// SIMATIC S7-200 project (STEP 7-Micro/WIN), CPU 224 CN REL 02.01

ORGANIZATION_BLOCK 主程序:OB1
TITLE=程序注释
BEGIN
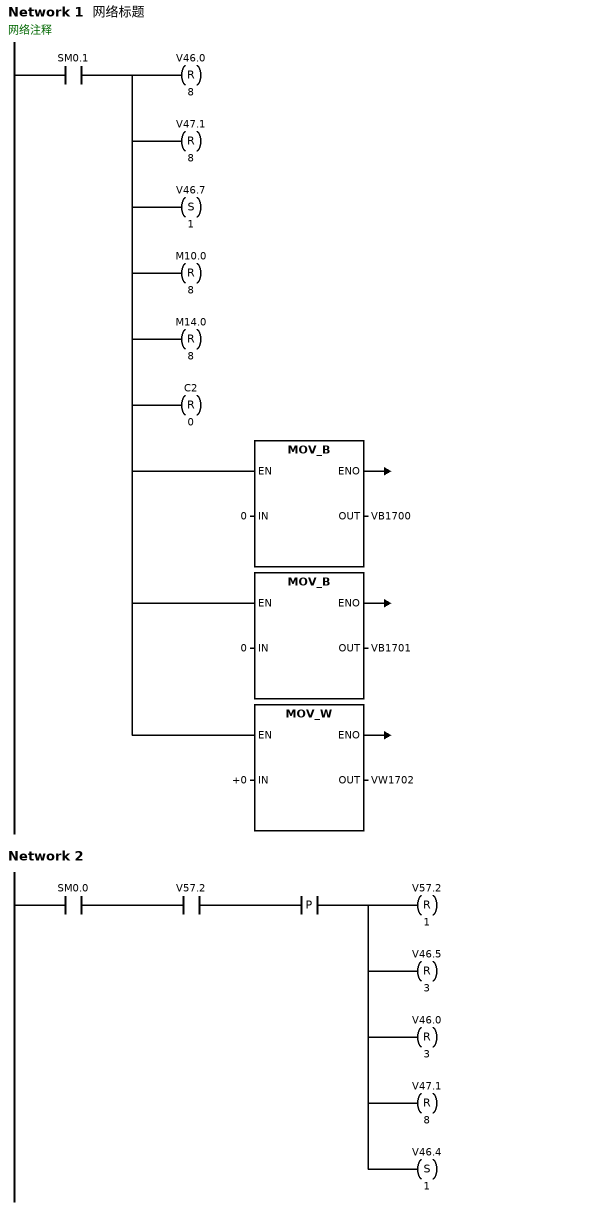
Network 1 // 网络标题
// 网络注释
LD     SM0.1
R      V46.0, 8
R      V47.1, 8
S      V46.7, 1
R      M10.0, 8
R      M14.0, 8
R      C2, 0
MOVB   0, VB1700
MOVB   0, VB1701
MOVW   +0, VW1702
Network 2
LD     SM0.0
A      V57.2
EU
R      V57.2, 1
R      V46.5, 3
R      V46.0, 3
R      V47.1, 8
S      V46.4, 1
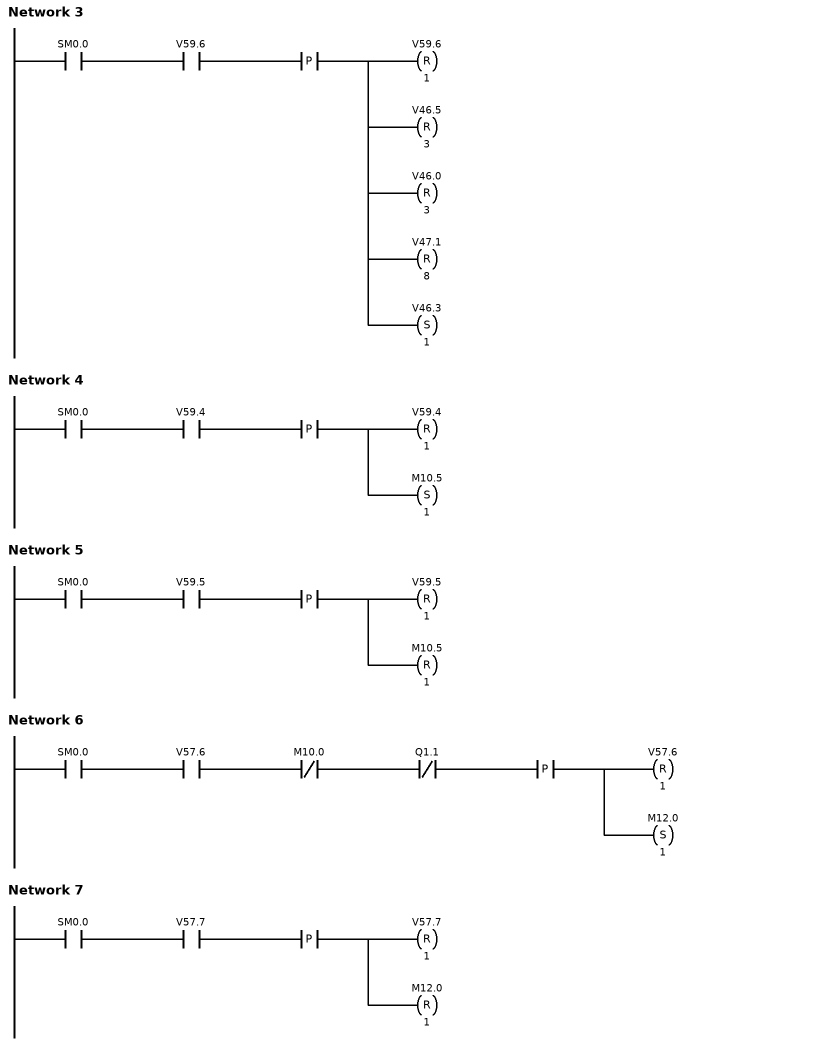
Network 3
LD     SM0.0
A      V59.6
EU
R      V59.6, 1
R      V46.5, 3
R      V46.0, 3
R      V47.1, 8
S      V46.3, 1
Network 4
LD     SM0.0
A      V59.4
EU
R      V59.4, 1
S      M10.5, 1
Network 5
LD     SM0.0
A      V59.5
EU
R      V59.5, 1
R      M10.5, 1
Network 6
LD     SM0.0
A      V57.6
AN     M10.0
AN     Q1.1
EU
R      V57.6, 1
S      M12.0, 1
Network 7
LD     SM0.0
A      V57.7
EU
R      V57.7, 1
R      M12.0, 1
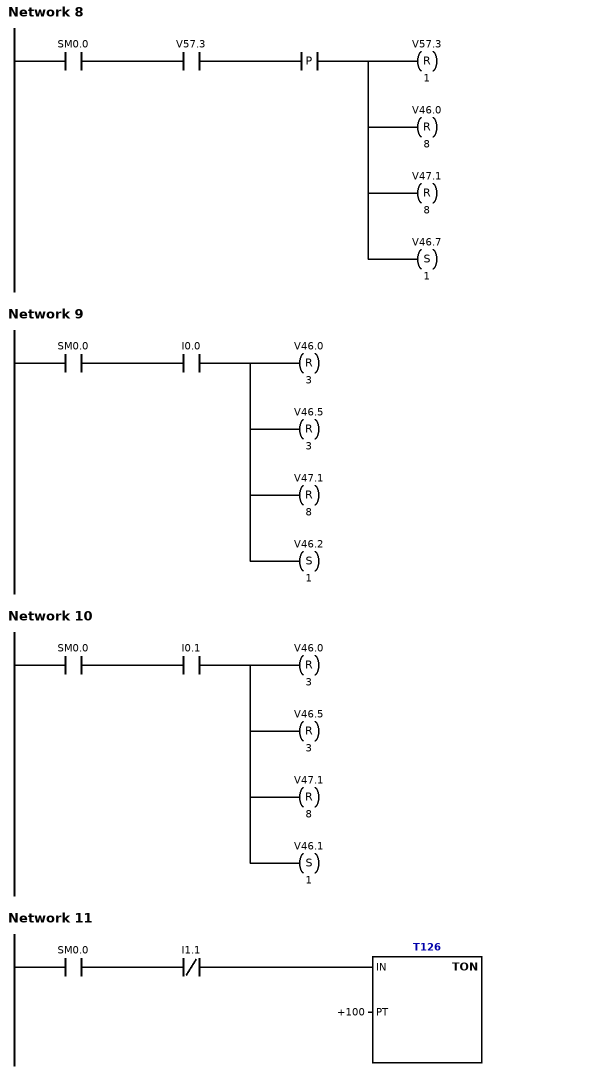
Network 8
LD     SM0.0
A      V57.3
EU
R      V57.3, 1
R      V46.0, 8
R      V47.1, 8
S      V46.7, 1
Network 9
LD     SM0.0
A      I0.0
R      V46.0, 3
R      V46.5, 3
R      V47.1, 8
S      V46.2, 1
Network 10
LD     SM0.0
A      I0.1
R      V46.0, 3
R      V46.5, 3
R      V47.1, 8
S      V46.1, 1
Network 11
LD     SM0.0
AN     I1.1
TON    T126, +100
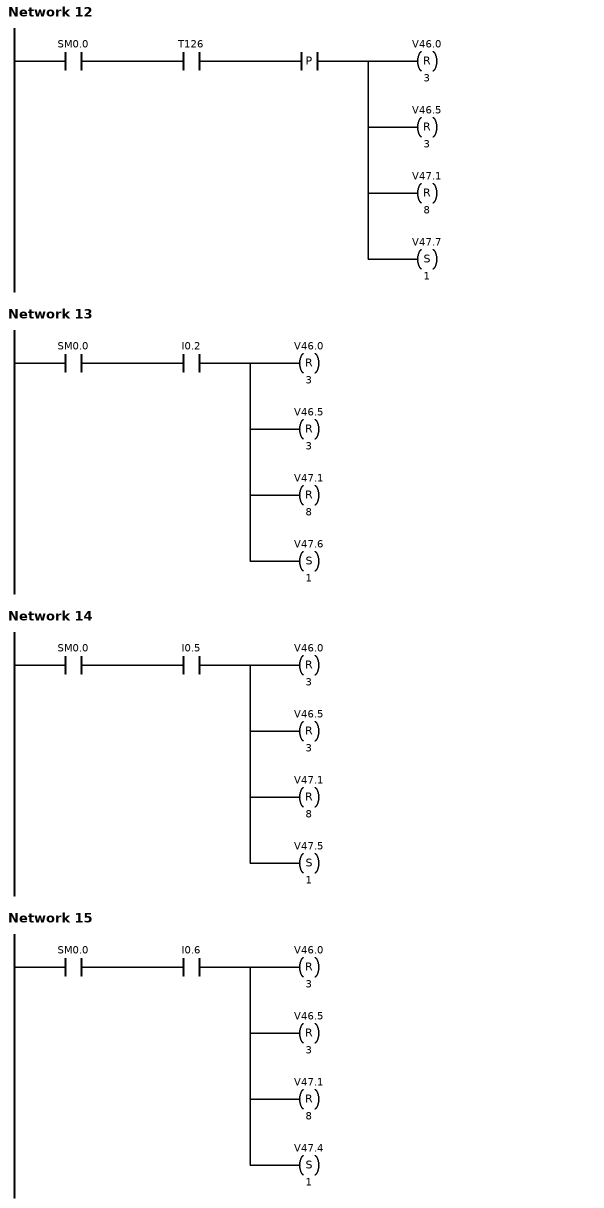
Network 12
LD     SM0.0
A      T126
EU
R      V46.0, 3
R      V46.5, 3
R      V47.1, 8
S      V47.7, 1
Network 13
LD     SM0.0
A      I0.2
R      V46.0, 3
R      V46.5, 3
R      V47.1, 8
S      V47.6, 1
Network 14
LD     SM0.0
A      I0.5
R      V46.0, 3
R      V46.5, 3
R      V47.1, 8
S      V47.5, 1
Network 15
LD     SM0.0
A      I0.6
R      V46.0, 3
R      V46.5, 3
R      V47.1, 8
S      V47.4, 1
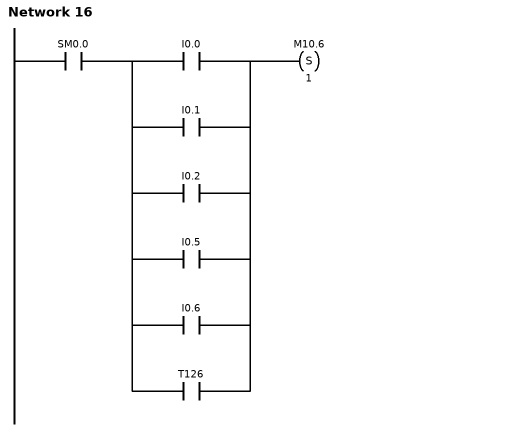
Network 16
LD     SM0.0
LD     I0.0
O      I0.1
O      I0.2
O      I0.5
O      I0.6
O      T126
ALD
S      M10.6, 1
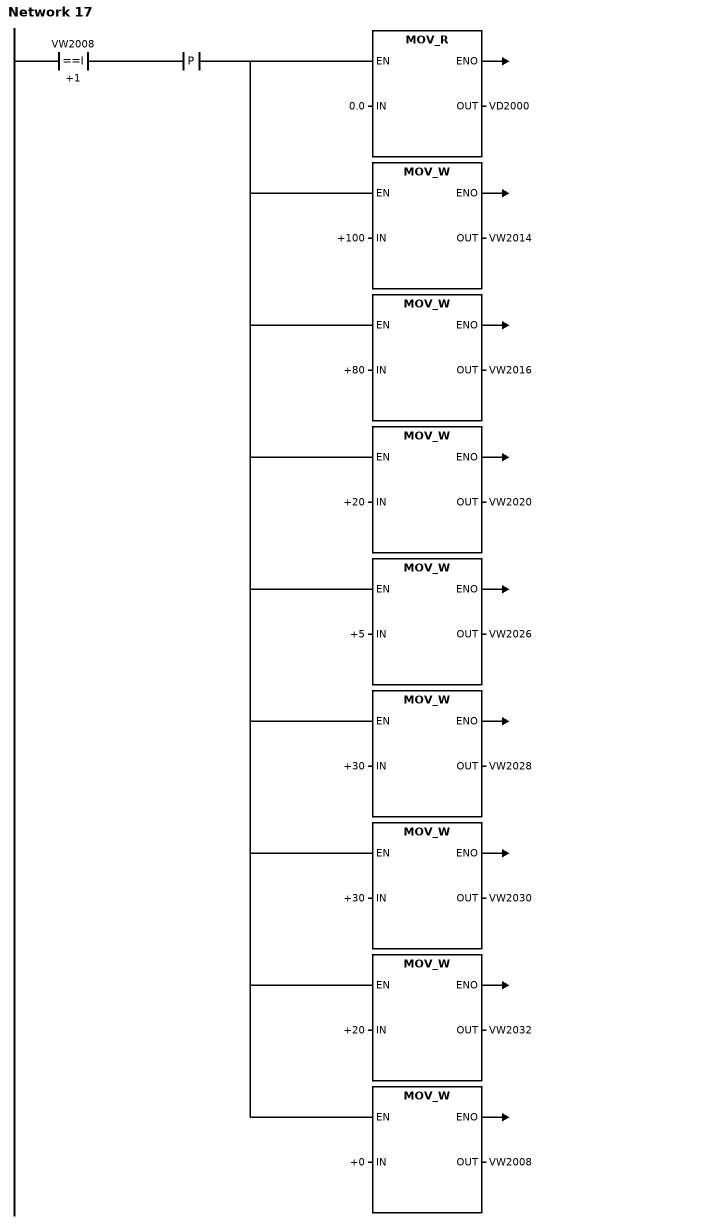
Network 17
LDW=   VW2008, +1
EU
MOVR   0.0, VD2000
MOVW   +100, VW2014
MOVW   +80, VW2016
MOVW   +20, VW2020
MOVW   +5, VW2026
MOVW   +30, VW2028
MOVW   +30, VW2030
MOVW   +20, VW2032
MOVW   +0, VW2008
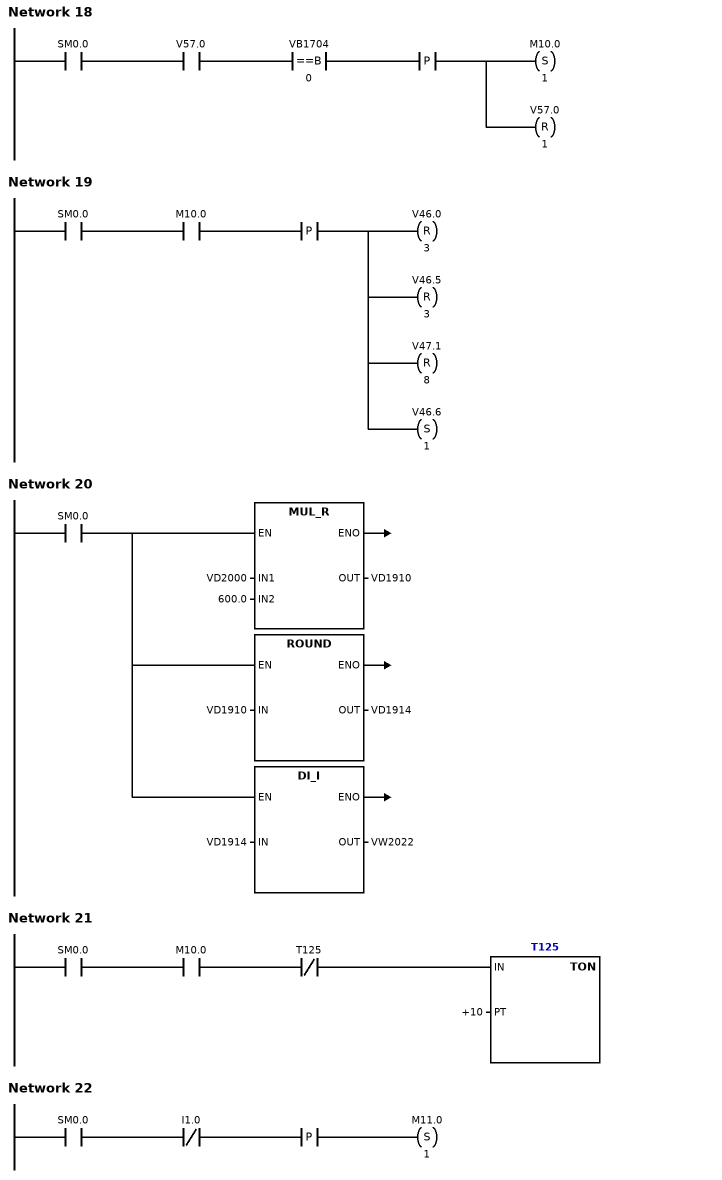
Network 18
LD     SM0.0
A      V57.0
AB=    VB1704, 0
EU
S      M10.0, 1
R      V57.0, 1
Network 19
LD     SM0.0
A      M10.0
EU
R      V46.0, 3
R      V46.5, 3
R      V47.1, 8
S      V46.6, 1
Network 20
LD     SM0.0
MOVR   VD2000, VD1910
*R     600.0, VD1910
ROUND  VD1910, VD1914
DTI    VD1914, VW2022
Network 21
LD     SM0.0
A      M10.0
AN     T125
TON    T125, +10
Network 22
LD     SM0.0
AN     I1.0
EU
S      M11.0, 1
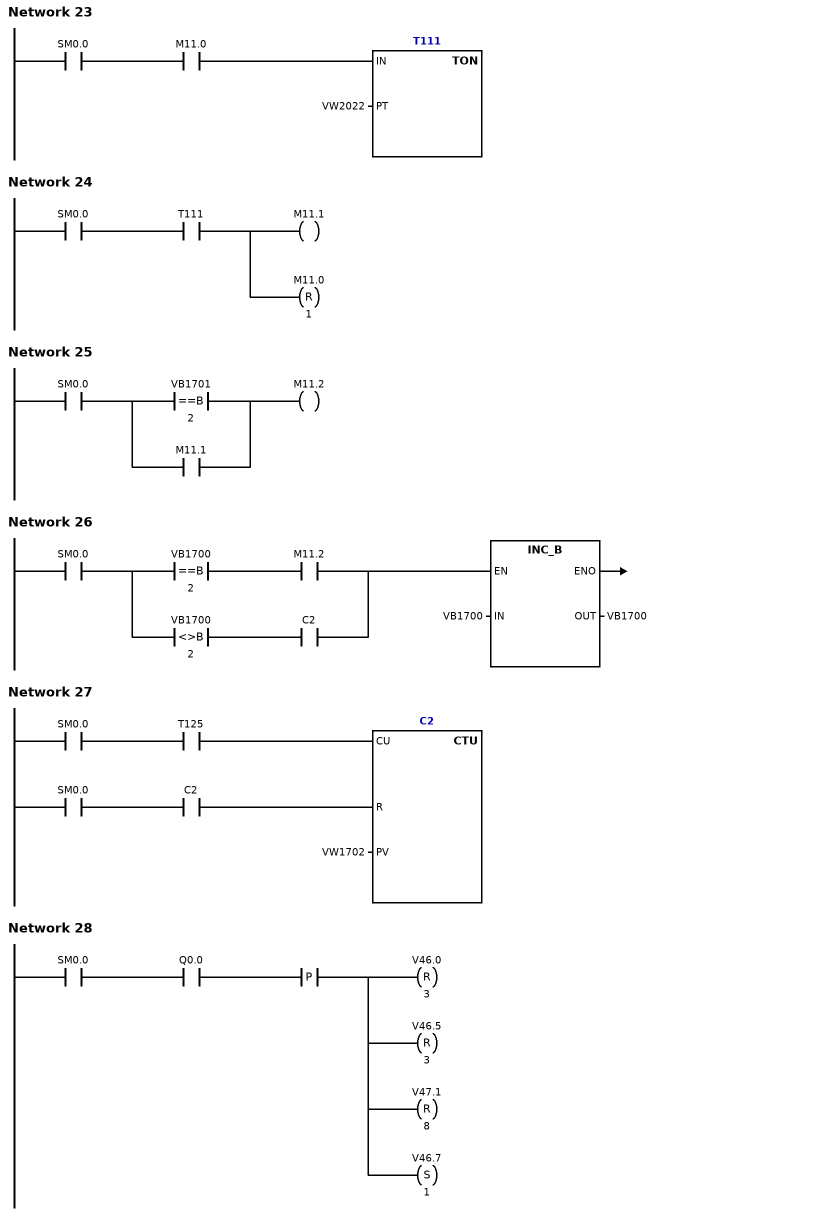
Network 23
LD     SM0.0
A      M11.0
TON    T111, VW2022
Network 24
LD     SM0.0
A      T111
=      M11.1
R      M11.0, 1
Network 25
LD     SM0.0
LDB=   VB1701, 2
O      M11.1
ALD
=      M11.2
Network 26
LD     SM0.0
LDB=   VB1700, 2
A      M11.2
LDB<>  VB1700, 2
A      C2
OLD
ALD
INCB   VB1700
Network 27
LD     SM0.0
A      T125
LD     SM0.0
A      C2
CTU    C2, VW1702
Network 28
LD     SM0.0
A      Q0.0
EU
R      V46.0, 3
R      V46.5, 3
R      V47.1, 8
S      V46.7, 1
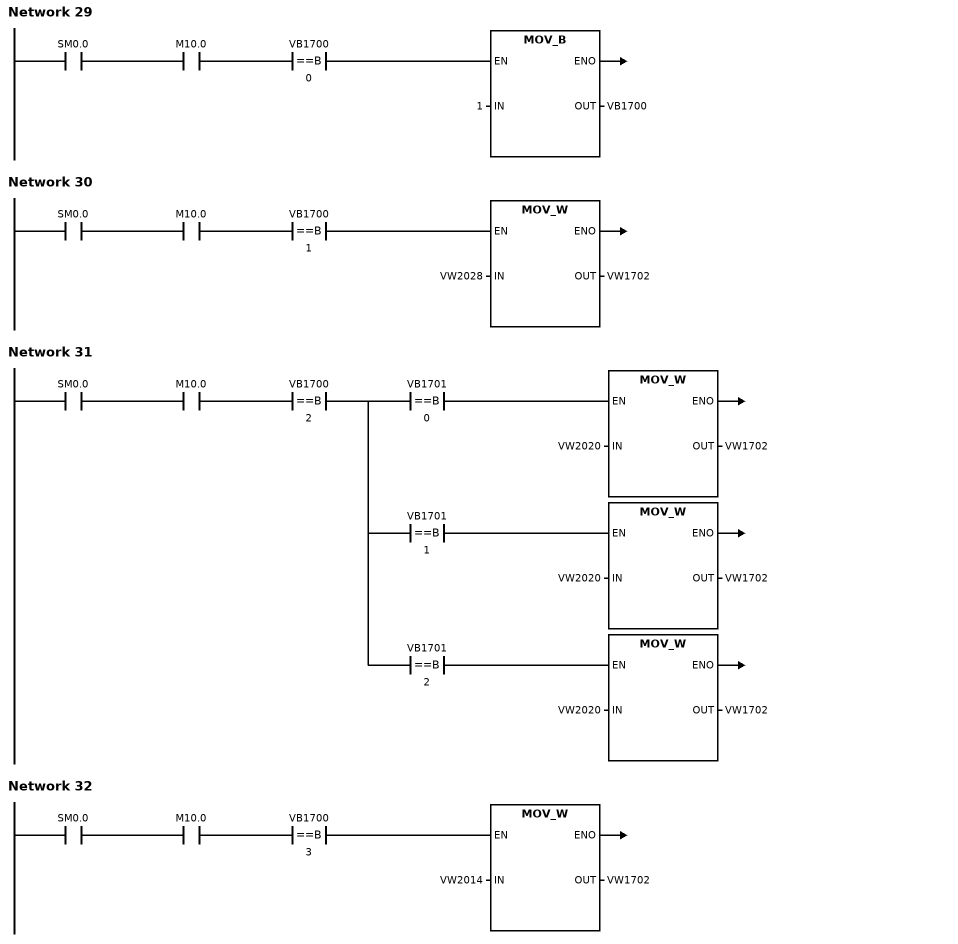
Network 29
LD     SM0.0
A      M10.0
AB=    VB1700, 0
MOVB   1, VB1700
Network 30
LD     SM0.0
A      M10.0
AB=    VB1700, 1
MOVW   VW2028, VW1702
Network 31
LD     SM0.0
A      M10.0
AB=    VB1700, 2
LPS
AB=    VB1701, 0
MOVW   VW2020, VW1702
LRD
AB=    VB1701, 1
MOVW   VW2020, VW1702
LPP
AB=    VB1701, 2
MOVW   VW2020, VW1702
Network 32
LD     SM0.0
A      M10.0
AB=    VB1700, 3
MOVW   VW2014, VW1702
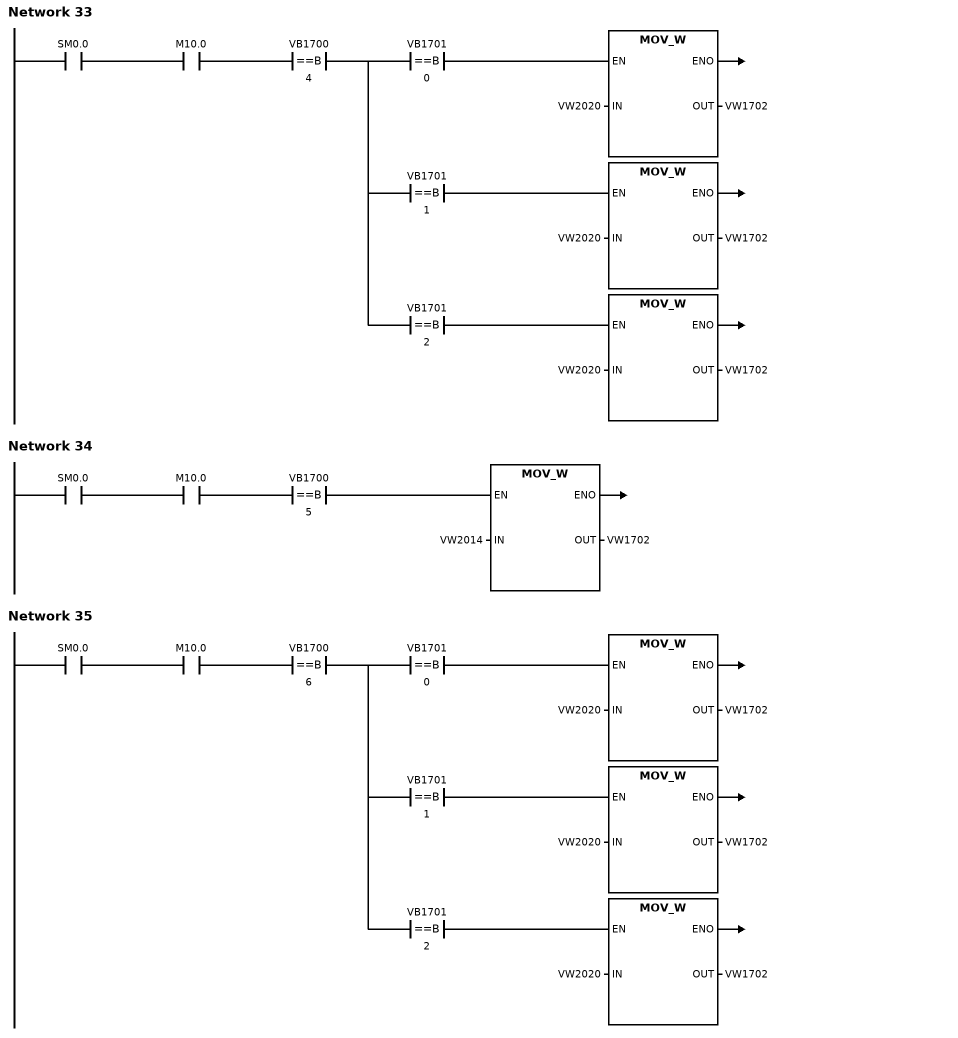
Network 33
LD     SM0.0
A      M10.0
AB=    VB1700, 4
LPS
AB=    VB1701, 0
MOVW   VW2020, VW1702
LRD
AB=    VB1701, 1
MOVW   VW2020, VW1702
LPP
AB=    VB1701, 2
MOVW   VW2020, VW1702
Network 34
LD     SM0.0
A      M10.0
AB=    VB1700, 5
MOVW   VW2014, VW1702
Network 35
LD     SM0.0
A      M10.0
AB=    VB1700, 6
LPS
AB=    VB1701, 0
MOVW   VW2020, VW1702
LRD
AB=    VB1701, 1
MOVW   VW2020, VW1702
LPP
AB=    VB1701, 2
MOVW   VW2020, VW1702
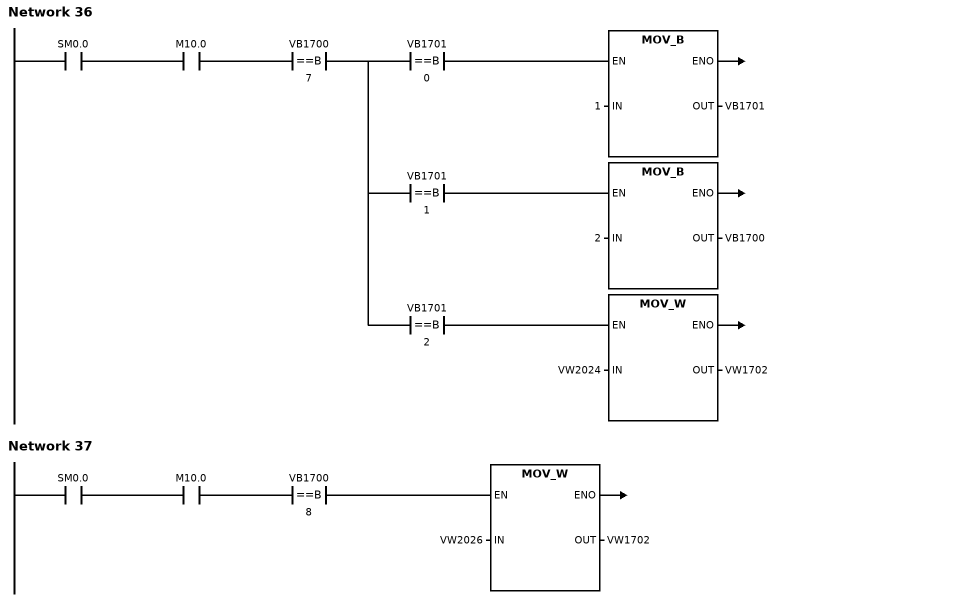
Network 36
LD     SM0.0
A      M10.0
AB=    VB1700, 7
LPS
AB=    VB1701, 0
MOVB   1, VB1701
LRD
AB=    VB1701, 1
MOVB   2, VB1700
LPP
AB=    VB1701, 2
MOVW   VW2024, VW1702
Network 37
LD     SM0.0
A      M10.0
AB=    VB1700, 8
MOVW   VW2026, VW1702
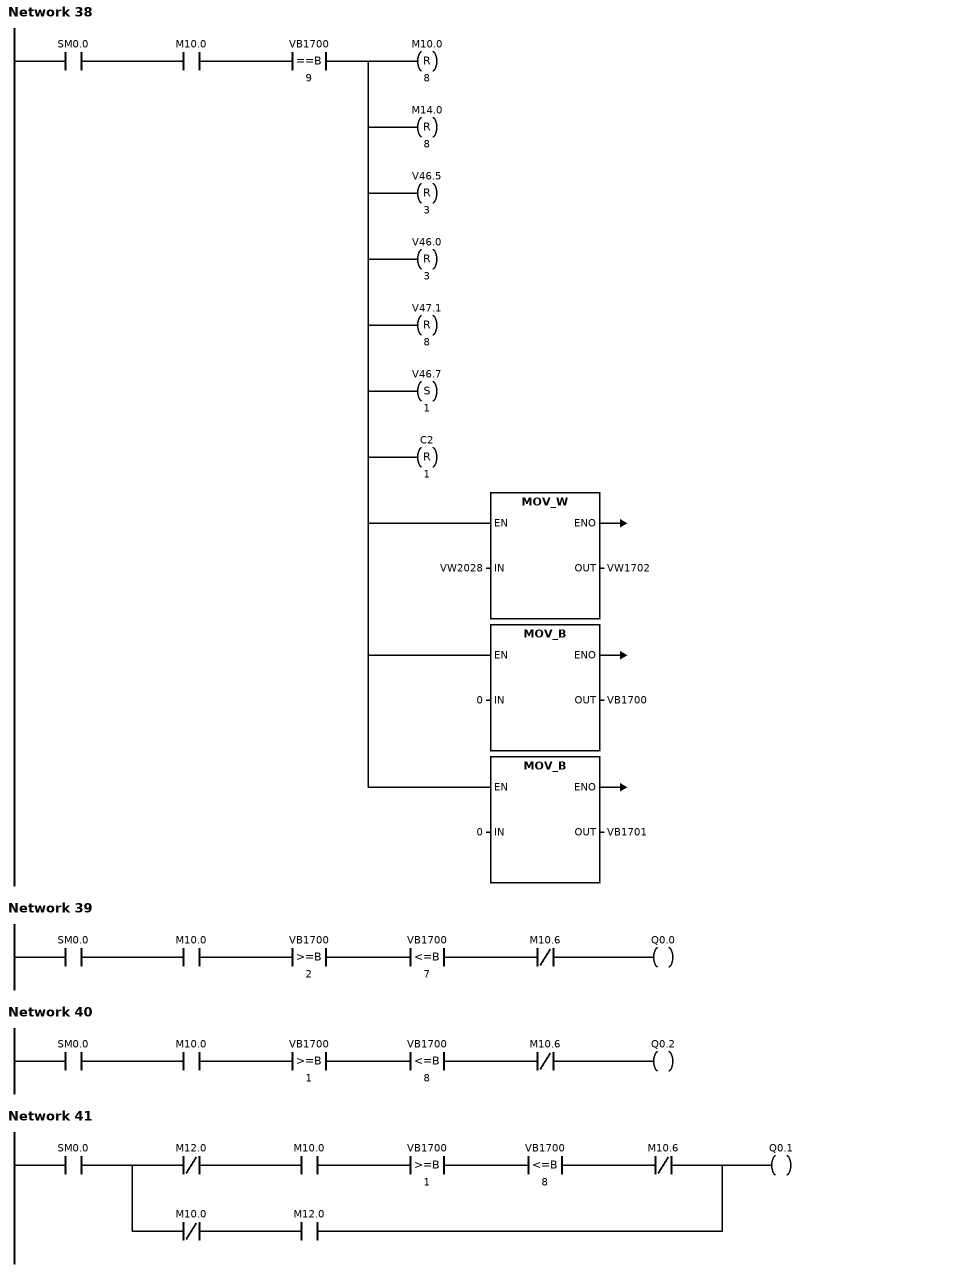
Network 38
LD     SM0.0
A      M10.0
AB=    VB1700, 9
R      M10.0, 8
R      M14.0, 8
R      V46.5, 3
R      V46.0, 3
R      V47.1, 8
S      V46.7, 1
R      C2, 1
MOVW   VW2028, VW1702
MOVB   0, VB1700
MOVB   0, VB1701
Network 39
LD     SM0.0
A      M10.0
AB>=   VB1700, 2
AB<=   VB1700, 7
AN     M10.6
=      Q0.0
Network 40
LD     SM0.0
A      M10.0
AB>=   VB1700, 1
AB<=   VB1700, 8
AN     M10.6
=      Q0.2
Network 41
LD     SM0.0
LDN    M12.0
A      M10.0
AB>=   VB1700, 1
AB<=   VB1700, 8
AN     M10.6
LDN    M10.0
A      M12.0
OLD
ALD
=      Q0.1
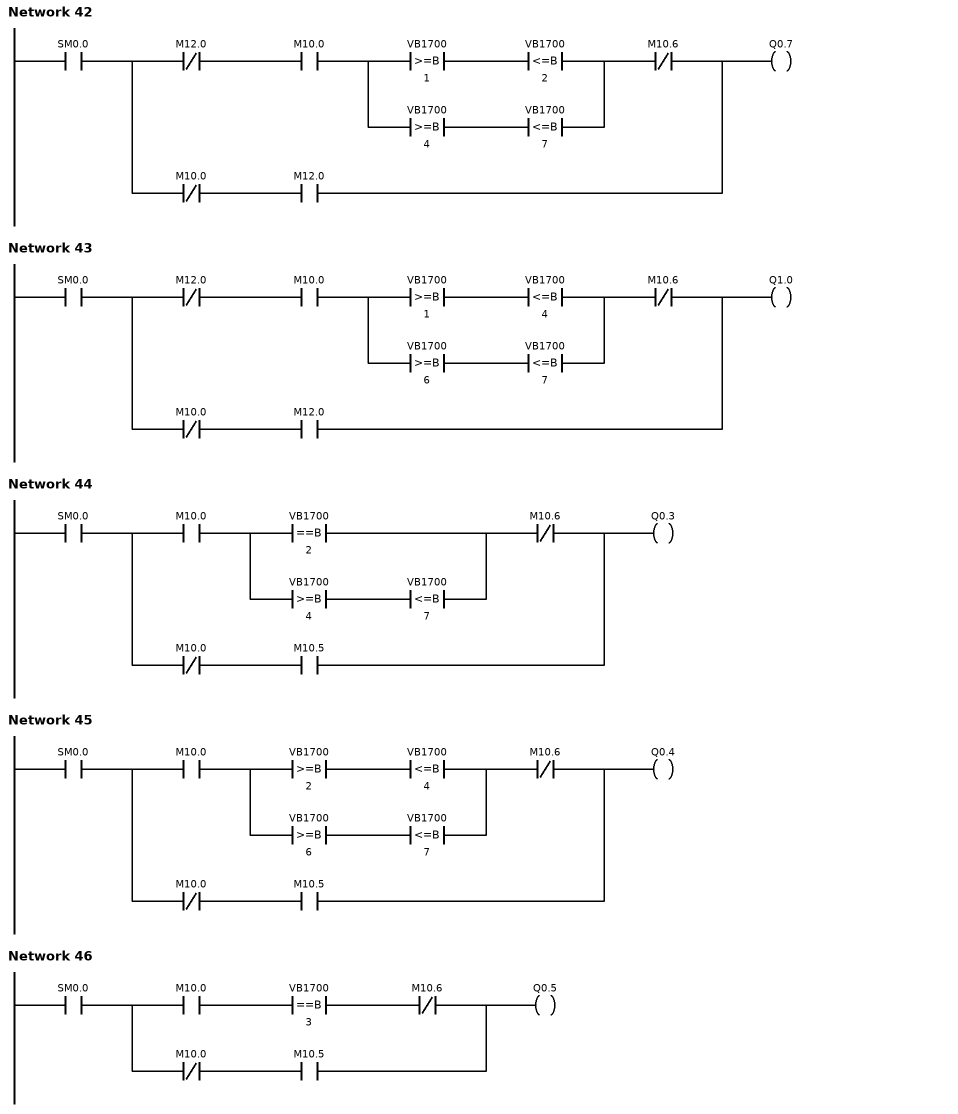
Network 42
LD     SM0.0
LDN    M12.0
A      M10.0
LDB>=  VB1700, 1
AB<=   VB1700, 2
LDB>=  VB1700, 4
AB<=   VB1700, 7
OLD
ALD
AN     M10.6
LDN    M10.0
A      M12.0
OLD
ALD
=      Q0.7
Network 43
LD     SM0.0
LDN    M12.0
A      M10.0
LDB>=  VB1700, 1
AB<=   VB1700, 4
LDB>=  VB1700, 6
AB<=   VB1700, 7
OLD
ALD
AN     M10.6
LDN    M10.0
A      M12.0
OLD
ALD
=      Q1.0
Network 44
LD     SM0.0
LD     M10.0
LDB=   VB1700, 2
LDB>=  VB1700, 4
AB<=   VB1700, 7
OLD
ALD
AN     M10.6
LDN    M10.0
A      M10.5
OLD
ALD
=      Q0.3
Network 45
LD     SM0.0
LD     M10.0
LDB>=  VB1700, 2
AB<=   VB1700, 4
LDB>=  VB1700, 6
AB<=   VB1700, 7
OLD
ALD
AN     M10.6
LDN    M10.0
A      M10.5
OLD
ALD
=      Q0.4
Network 46
LD     SM0.0
LD     M10.0
AB=    VB1700, 3
AN     M10.6
LDN    M10.0
A      M10.5
OLD
ALD
=      Q0.5
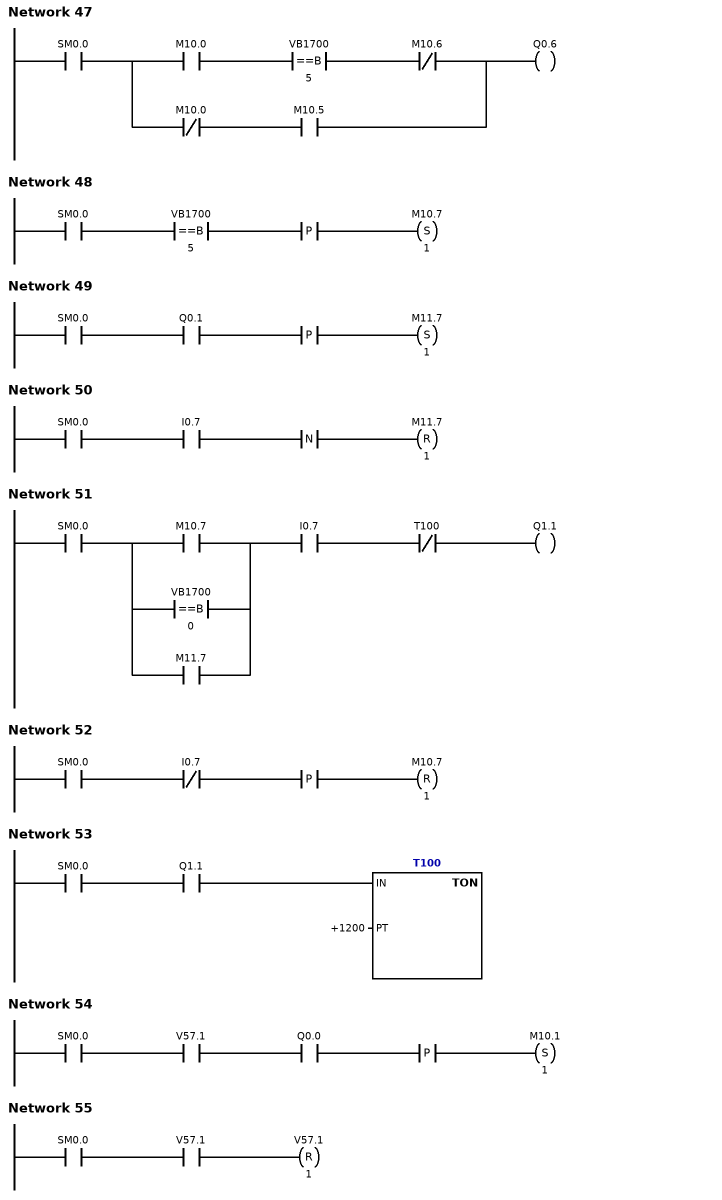
Network 47
LD     SM0.0
LD     M10.0
AB=    VB1700, 5
AN     M10.6
LDN    M10.0
A      M10.5
OLD
ALD
=      Q0.6
Network 48
LD     SM0.0
AB=    VB1700, 5
EU
S      M10.7, 1
Network 49
LD     SM0.0
A      Q0.1
EU
S      M11.7, 1
Network 50
LD     SM0.0
A      I0.7
ED
R      M11.7, 1
Network 51
LD     SM0.0
LD     M10.7
OB=    VB1700, 0
O      M11.7
ALD
A      I0.7
AN     T100
=      Q1.1
Network 52
LD     SM0.0
AN     I0.7
EU
R      M10.7, 1
Network 53
LD     SM0.0
A      Q1.1
TON    T100, +1200
Network 54
LD     SM0.0
A      V57.1
A      Q0.0
EU
S      M10.1, 1
Network 55
LD     SM0.0
A      V57.1
R      V57.1, 1
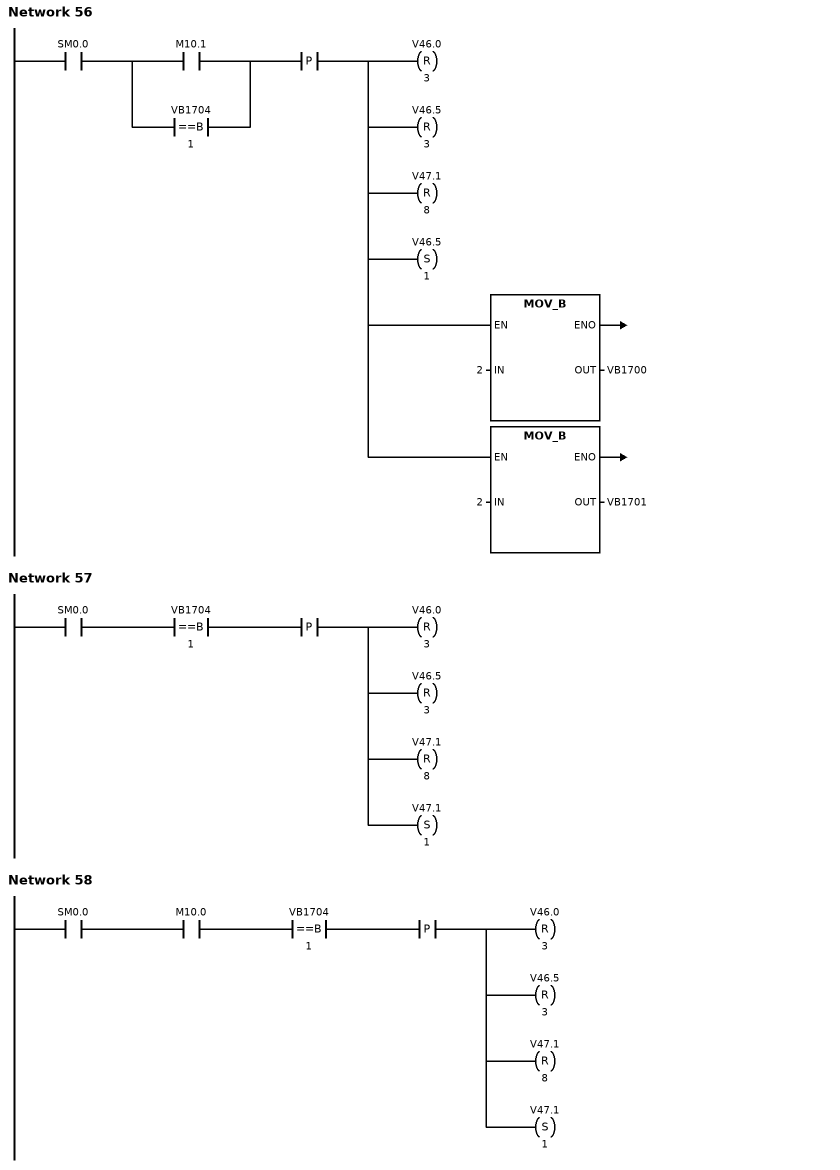
Network 56
LD     SM0.0
LD     M10.1
OB=    VB1704, 1
ALD
EU
R      V46.0, 3
R      V46.5, 3
R      V47.1, 8
S      V46.5, 1
MOVB   2, VB1700
MOVB   2, VB1701
Network 57
LD     SM0.0
AB=    VB1704, 1
EU
R      V46.0, 3
R      V46.5, 3
R      V47.1, 8
S      V47.1, 1
Network 58
LD     SM0.0
A      M10.0
AB=    VB1704, 1
EU
R      V46.0, 3
R      V46.5, 3
R      V47.1, 8
S      V47.1, 1
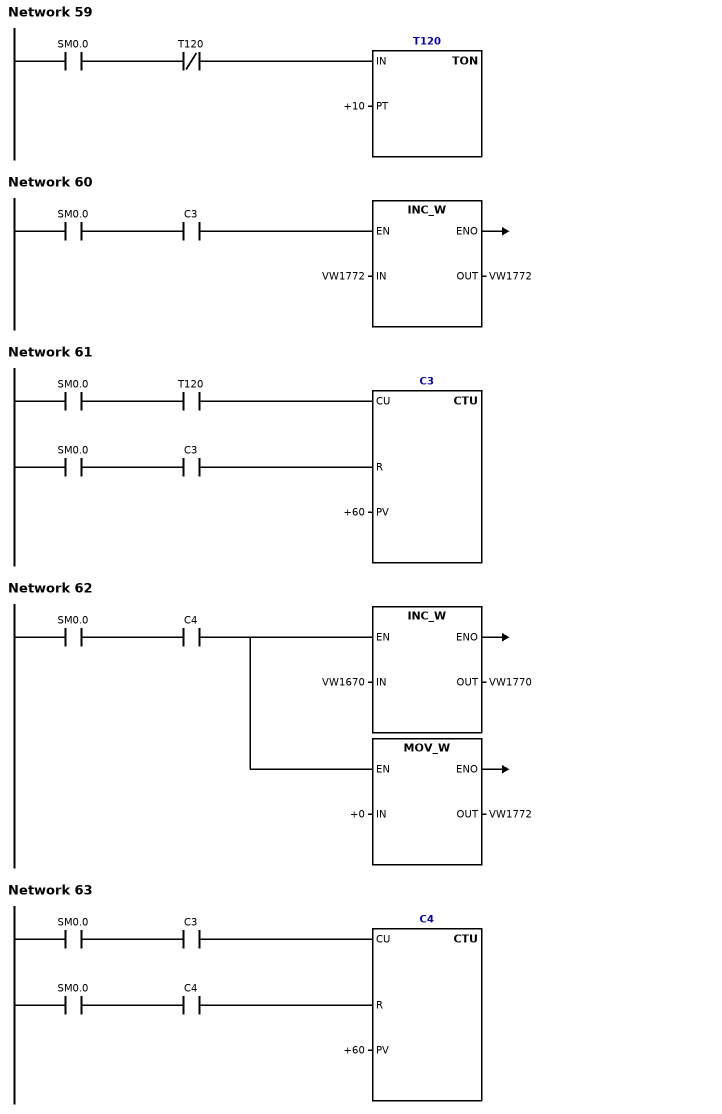
Network 59
LD     SM0.0
AN     T120
TON    T120, +10
Network 60
LD     SM0.0
A      C3
INCW   VW1772
Network 61
LD     SM0.0
A      T120
LD     SM0.0
A      C3
CTU    C3, +60
Network 62
LD     SM0.0
A      C4
MOVW   VW1670, VW1770
INCW   VW1770
MOVW   +0, VW1772
Network 63
LD     SM0.0
A      C3
LD     SM0.0
A      C4
CTU    C4, +60
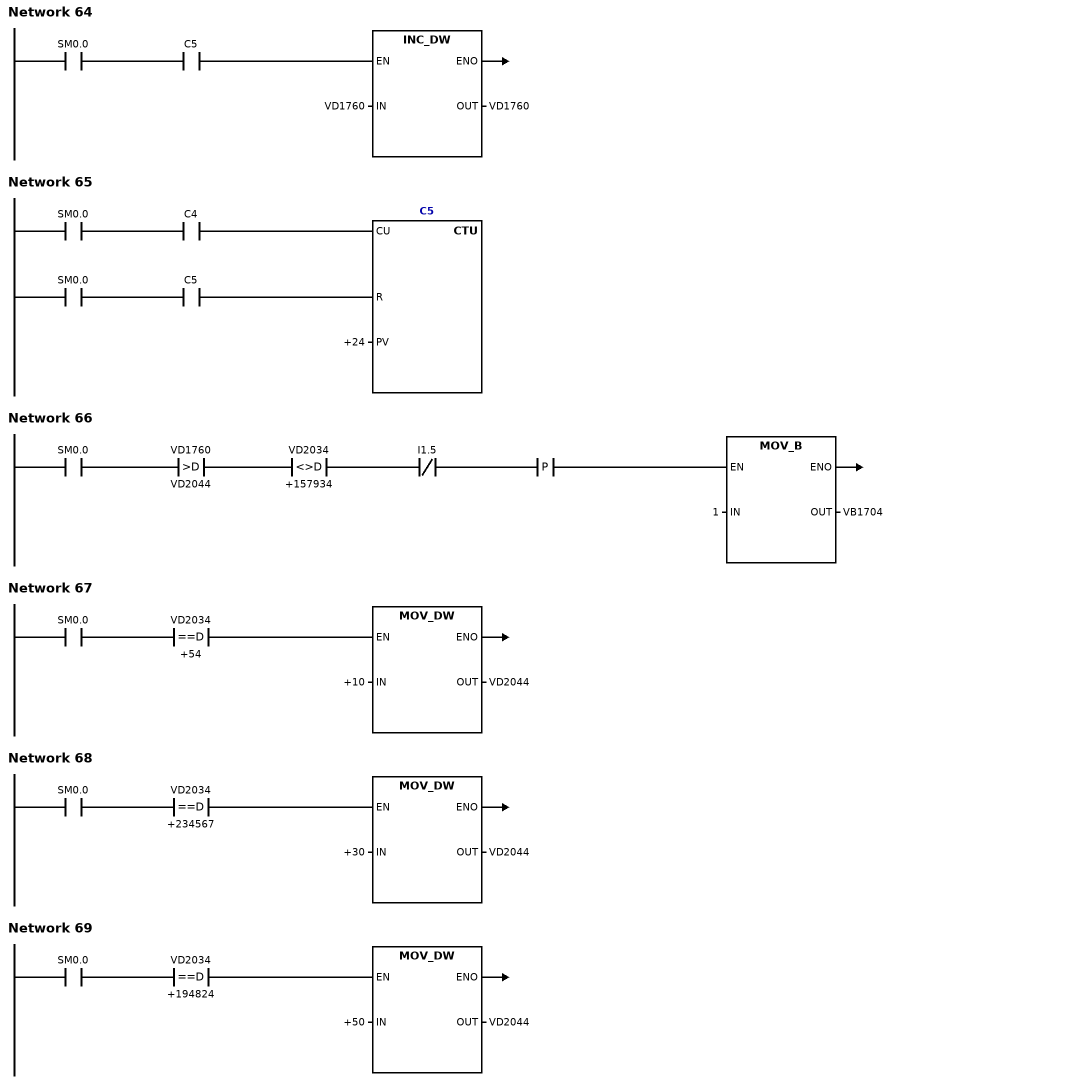
Network 64
LD     SM0.0
A      C5
INCD   VD1760
Network 65
LD     SM0.0
A      C4
LD     SM0.0
A      C5
CTU    C5, +24
Network 66
LD     SM0.0
AD>    VD1760, VD2044
AD<>   VD2034, +157934
AN     I1.5
EU
MOVB   1, VB1704
Network 67
LD     SM0.0
AD=    VD2034, +54
MOVD   +10, VD2044
Network 68
LD     SM0.0
AD=    VD2034, +234567
MOVD   +30, VD2044
Network 69
LD     SM0.0
AD=    VD2034, +194824
MOVD   +50, VD2044
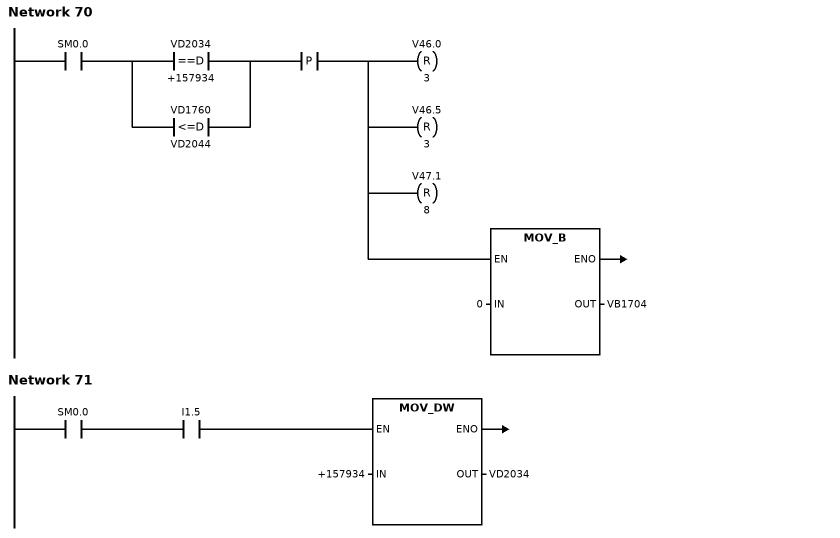
Network 70
LD     SM0.0
LDD=   VD2034, +157934
OD<=   VD1760, VD2044
ALD
EU
R      V46.0, 3
R      V46.5, 3
R      V47.1, 8
MOVB   0, VB1704
Network 71
LD     SM0.0
A      I1.5
MOVD   +157934, VD2034
END_ORGANIZATION_BLOCK

// SBR1: protected block, not included

// SBR2: protected block, not included

// (further data pages could not be read)
